(* IEC 61131-3 sources: plc-tank-filling-station/src, 2 files *)

(* ---- E_TankState.st ---- *)
{attribute 'qualified_only'}
{attribute 'strict'}
TYPE E_TankState :
(
    IDLE     := 0,
    FILLING  := 1,
    MIXING   := 2,
    DRAINING := 3,
    COMPLETE := 4,
    FAULT    := 5
);
END_TYPE

(* ---- PLC_PRG.st ---- *)
PROGRAM PLC_PRG

VAR
    xStart          : BOOL;
    xReset          : BOOL;
    xEmergencyStop  : BOOL;

    fbTank          : FB_TankController;
    fbSimulation    : FB_TankSimulation;
END_VAR

fbTank(
    xStart         := xStart,
    xReset         := xReset,
    xEmergencyStop := xEmergencyStop,
    fLevelPercent  := fbSimulation.fLevelPercent
);

fbSimulation(
    xInletValve := fbTank.xInletValve,
    xDrainValve := fbTank.xDrainValve
);
END_PROGRAM
